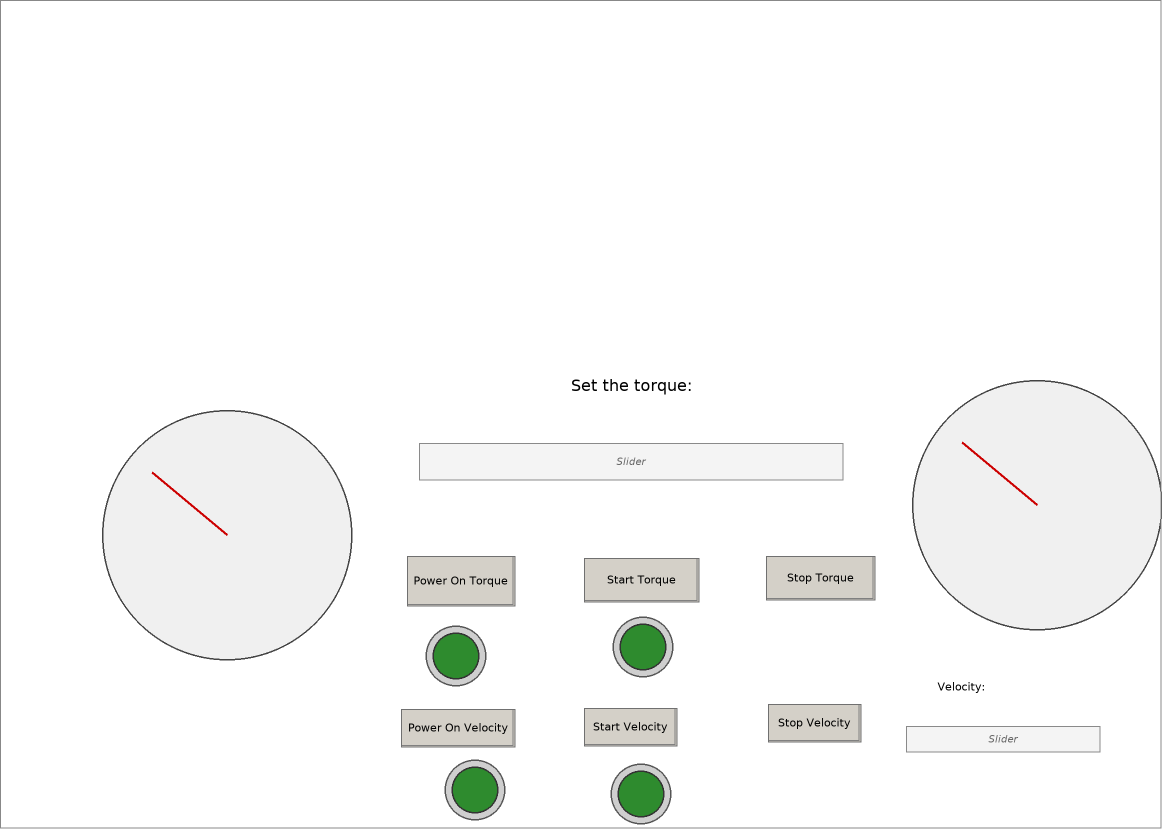
VISUALIZATION Visualization  // 1162x829
    Slider (419,443 424x37), variable: MAIN.TVAL, scale 0..100
    Button (584,558 115x44), "Start Torque"
        OnMouseClick: toggle MAIN.Start1Btn
    Button (407,556 108x50), "Power On Torque"
        OnMouseClick: toggle MAIN.PowerOnTorqueBtn
    Button (766,556 109x44), "Stop Torque"
        OnMouseClick: toggle MAIN.Stop1Btn
    Label (532,358 200x55), "Set the torque:"
    Button (401,709 114x38), "Power On Velocity"
        OnMouseClick: toggle Velocity.PowerOnVelocityBtn
    Button (584,708 93x38), "Start Velocity"
        OnMouseClick: toggle Velocity.Start2Btn
    Button (768,704 93x38), "Stop Velocity"
        OnMouseClick: toggle Velocity.Stop2Btn
    Meter360 (102,410 250x250), value: Actual_Velocity, style: Meter-Meter360-Gray, scale format: %.1f, scale 0..2000
    Label (899,667 125x40), "Velocity:"
    Meter360 (912,380 250x250), value: ActualTorque, style: Meter-Meter360-Gray, scale format: %.1f, scale 0..12
    Lamp1 (421,621 70x70), variable: MAIN.Power1_Active, style: Lamp-Lamp1-Green
    Lamp1 (608,612 70x70), variable: MAIN.TorqueEnable, style: Lamp-Lamp1-Green
    Lamp1 (606,759 70x70), variable: Velocity.MV2_InVelocity, style: Lamp-Lamp1-Green
    Lamp1 (440,755 70x70), variable: Velocity.Power2_Active, style: Lamp-Lamp1-Green
    Slider (906,726 194x26), variable: Velocity.MVelocity, scale 0..1000
END_VISUALIZATION

(* stored: Version 1.1.0.1, ProductVersion 3.1.4024.4
   Visu Visualization: Id {191cc02f-e427-402b-9629-de7e1be62d0e} *)
